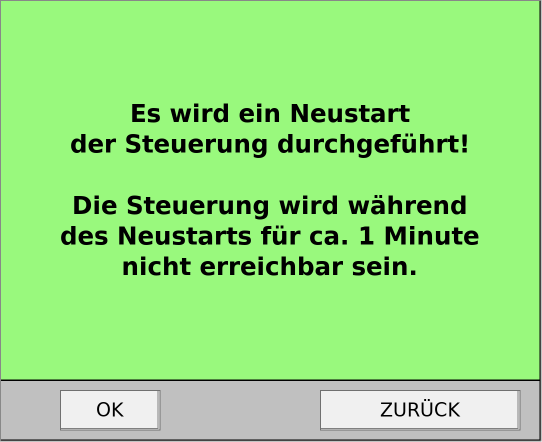
VISUALIZATION V_TCReset  // 542x442
vAR_IN_OUT
	
END_VAR
    Rectangle (0,380 540x60)
    Button (60,390 100x40), "OK"
        OnMouseUp: change screen: Previous 
        OnMouseDown: toggle gfbSystemCX.VbTCReset
    Button (320,390 200x40), "ZURÜCK"
        OnMouseUp: change screen: Previous 
    Rectangle (0,0 540x380), "Es wird ein Neustart der Steuerung durchgeführt! Die Steuerung wird während des Neustarts für ca. 1 Minute nicht erreichbar sein."
END_VISUALIZATION

(* stored: Version 1.1.0.1, ProductVersion 3.1.4018.10
   Visu V_TCReset: Id {5888a373-99ff-4aab-81ff-d513e99b70a6} *)
